FUNCTION_BLOCK Dimmer
VAR_INPUT
	input01: BOOL;
	input02: BOOL;
END_VAR
VAR_OUTPUT
	output: INT;
END_VAR
VAR
	tonLongPress_01: TON;
	tonLongPress_02: TON;
	step: INT;
	dimmer_perc: REAL;

	rampUp: RampUp;
	rampDown: RampDown;
END_VAR


	
CASE step OF
	0:	//	Key pressed
		IF input01 THEN
			step := 10;
		ELSIF input02 THEN
			step := 50;	
		END_IF
		rampUp(Enable := FALSE);
		rampDown(Enable := FALSE);
		tonLongPress_01(IN := FALSE);
		tonLongPress_02(IN := FALSE);
		
		
	10:	//	Short Press - On
		tonLongPress_01(IN:= input01, PT:= T_LONG_PRESS, Q=> , ET=> );
		IF tonLongPress_01.Q THEN
			step :=	20;
		ELSIF (NOT input01) THEN
			dimmer_perc	:=	100;
			step		:=	0;
		END_IF
	
	20: // Long Press - Up
		rampUp(
			Setpoint:= 100, 
			RampUpTime:= RAMP_UP_TIME, 
			Enable:= TRUE, 
			Output=> dimmer_perc, 
			InProgress=> );
			
		IF (NOT input01) THEN
			step	:=	0;
		END_IF
	

	50:	//	Short press - Off
		tonLongPress_02(IN:= input02, PT:= T_LONG_PRESS, Q=> , ET=> );
		IF tonLongPress_02.Q THEN
			step :=	60;
		ELSIF (NOT input02) THEN
			dimmer_perc	:=	0;
			step		:=	0;
		END_IF
	
	60:	//	Long press - Down
		rampDown(
			Setpoint:= 0, 
			RampDownTime:= RAMP_DOWN_TIME, 
			Enable:= TRUE, 
			Output=> dimmer_perc, 
			InProgress=> );
		
		IF (NOT input02) THEN
			step	:=	0;
		END_IF
	
END_CASE

	output	:=	REAL_TO_INT(F_Scaling(
								Variable_In:= dimmer_perc, 
								ZeroIn:= 0, 
								ZeroOut:= 100, 
								SpanIn:= 0, 
								SpanOut:= 32767));

END_FUNCTION_BLOCK

(* stored: Version 1.1.0.1, ProductVersion 3.1.4024.13
   POU Dimmer: Id {72de836e-7852-4ce8-a2be-acbaaea23600}, SpecialFunc None *)
